// TIA Portal V16 export
// export: Created 2024-09-05T17:40:13.9890551Z, ExportSetting WithDefaults, DisplayName Totally Integrated Automation Portal, DisplayVersion V16 Update 6, DisplayName TIA Portal Version Control Interface, DisplayVersion V16 Update 2, DisplayName TIA Portal Openness, DisplayVersion V16 Update 6, DisplayName STEP 7 Professional, DisplayVersion V16 Update 6, DisplayName STEP 7 Safety, DisplayVersion V16, DisplayName WinCC Advanced, DisplayVersion V16 Update 6
TYPE "UDT_Camera_Keyence_IV"
// stored: IsFailsafeCompliant false
   STRUCT
      ProgramNumber : SInt;
      Start : Bool;
      Done : Bool;
      ResultReadyAfterChange : Bool;
      Result : Int;
      ProgramOK : Bool;
      ProgramChangeNOK : Bool;
      Attempts : Int;
      MinOKAtempts : Int;
      Tool : Array[1..16] of Bool;
   END_STRUCT;
END_TYPE
